ABB RobotStudio station: step_smartcomponet.rspag

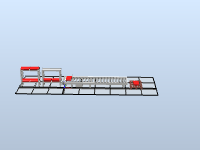
--- station ---
Station step_smartcomponet (saved by RobotStudio 6.8.8307.1040)
Controller IRB_120_3kg_0.58m_3
  mechanical unit ROB_1: IRB120_3_58__01, 6 joints, base frame (0, 0, 0) mm
Layout (positions relative to the parent item):
  - IRB4600_60_205_C_01 [mechanism, from Robots\IRB4600_60_205_C_G_01.rslib] at (0, 0, 0) mm; joint values [0, 0, 0, 0, 0.5236, 0] (rad or m)
  - 950_4000_h2 [part, from Equipment\Conveyor 950 4000 h2.rslib]
  - CAJA [part, from Step_smartcomponet\SOLCAJA.rslib] at (-590.31, 450, 412.42) mm
  - SmartComponent_1 [smart component, from Step_smartcomponet\SmartComponent_1.rslib]
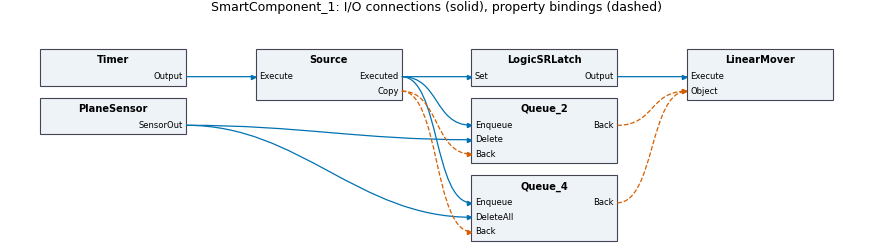
      connections:
        Timer.Output -> Source.Execute
        Source.Executed -> Queue_2.Enqueue
        LogicSRLatch.Output -> LinearMover.Execute
        PlaneSensor.SensorOut -> Queue_2.Delete
        Source.Executed -> Queue_4.Enqueue
        PlaneSensor.SensorOut -> Queue_4.DeleteAll
        Source.Executed -> LogicSRLatch.Set
        Source.Copy => Queue_2.Back
        Queue_2.Back => LinearMover.Object
        Source.Copy => Queue_4.Back
        Queue_4.Back => LinearMover.Object
    - Source [smart component, from Components\Source.rslib]
        properties: Source=CAJA1; Copy=(none); Parent=(none); Position=[3.9 0.5 0.4]; Orientation=[0 0 0]; Transient=true; PhysicsBehavior=0
    - Timer [smart component, from Components\Timer.rslib]
        properties: StartTime=0; Interval=7; Repeat=true; CurrentTime=256.632
    - LinearMover [smart component, from Components\LinearMover.rslib]
        properties: Object=(none); Direction=[-1 0 0]; Speed=0.6; Reference=Global; ReferenceObject=(none)
    - PlaneSensor [smart component, from Components\PlaneSensor.rslib]
        properties: Origin=[0.5 0.1 0.45]; Axis1=[0 0.2 0.3]; Axis2=[0 0.5 0]; SensedPart=(none)
      - _sensorPart_ [part, from Step_smartcomponet\SmartComponent_1.rslib]
    - LogicSRLatch [smart component, from Components\LogicSRLatch.rslib]
    - Queue_4 [smart component, from Components\Queue.rslib]
        properties: Back=(none); Front=(none); Queue={b297857b-f8dc-4992-8a1c-48ad92a09bcc}; NumberOfObjects=1
  - IRB120_3_58__01 [mechanism, from Robots\IRB120_3_58_G_01.rslib] at (0, 0, 0) mm; joint values [0, 0, 0, 0, 0.5236, 0] (rad or m)
  - Plant Shelf Assem [graphiccomponentgroup, from Step_smartcomponet\Stand de cajas vacio.rslib] at (-1309.51, 39.88, -195.16) mm, rotated rx 90 ry 0 rz 90 deg
    - Leg [part, from Step_smartcomponet\Stand de cajas vacio.rslib] at (58.14, 192.19, 978.34) mm, rotated rx 90 ry 0 rz 0 deg
    - Leg [part, from Step_smartcomponet\Stand de cajas vacio.rslib] at (432.79, 192.19, 978.34) mm, rotated rx 90 ry 0 rz 0 deg
    - Leg [part, from Step_smartcomponet\Stand de cajas vacio.rslib] at (58.14, 192.19, -151.96) mm, rotated rx 90 ry 0 rz 0 deg
    - Leg [part, from Step_smartcomponet\Stand de cajas vacio.rslib] at (432.79, 192.19, -151.96) mm, rotated rx 90 ry 0 rz 0 deg
    - Bottom Support Beam [part, from Step_smartcomponet\Stand de cajas vacio.rslib] at (432.79, 395.39, 1016.44) mm, rotated rx 0 ry 90 rz 0 deg
    - Bottom Support Beam [part, from Step_smartcomponet\Stand de cajas vacio.rslib] at (432.79, 395.39, -63.06) mm, rotated rx 0 ry 90 rz 0 deg
    - Top Support Beam [part, from Step_smartcomponet\Stand de cajas vacio.rslib] at (432.79, 1271.69, -63.06) mm, rotated rx 0 ry 90 rz 0 deg
    - Top Support Beam [part, from Step_smartcomponet\Stand de cajas vacio.rslib] at (432.79, 1271.69, 1010.09) mm, rotated rx 0 ry 90 rz 0 deg
    - Shelf Platform [part, from Step_smartcomponet\Stand de cajas vacio.rslib] at (121.64, 1303.08, 1067.24) mm
    - Shelf Platform [part, from Step_smartcomponet\Stand de cajas vacio.rslib] at (216.89, 1303.44, 1067.24) mm
    - Shelf Platform [part, from Step_smartcomponet\Stand de cajas vacio.rslib] at (312.14, 1303.44, 1067.24) mm
    - Shelf Platform [part, from Step_smartcomponet\Stand de cajas vacio.rslib] at (432.79, 1303.44, 1067.24) mm, rotated rx 0 ry 0 rz 90 deg
    - Shelf Platform [part, from Step_smartcomponet\Stand de cajas vacio.rslib] at (96.24, 1398.69, 1067.24) mm, rotated rx 0 ry 0 rz -90 deg
    - Shelf Platform [part, from Step_smartcomponet\Stand de cajas vacio.rslib] at (121.64, 484.29, 1067.24) mm
    - Shelf Platform [part, from Step_smartcomponet\Stand de cajas vacio.rslib] at (216.89, 484.29, 1067.24) mm
    - Shelf Platform [part, from Step_smartcomponet\Stand de cajas vacio.rslib] at (312.14, 484.29, 1067.24) mm
    - Shelf Platform [part, from Step_smartcomponet\Stand de cajas vacio.rslib] at (96.24, 579.54, 1067.24) mm, rotated rx 0 ry 0 rz -90 deg
    - Shelf Platform [part, from Step_smartcomponet\Stand de cajas vacio.rslib] at (432.79, 484.29, 1067.24) mm, rotated rx 0 ry 0 rz 90 deg
    - Bracket [part, from Step_smartcomponet\Stand de cajas vacio.rslib] at (96.24, 395.39, -82.11) mm, rotated rx 90 ry 0 rz 0 deg
    - Bracket [part, from Step_smartcomponet\Stand de cajas vacio.rslib] at (96.24, 1271.69, -78.94) mm, rotated rx 90 ry 0 rz 0 deg
    - Bracket [part, from Step_smartcomponet\Stand de cajas vacio.rslib] at (432.79, 1271.69, -78.94) mm, rotated rx -90 ry 0 rz 180 deg
    - Bracket [part, from Step_smartcomponet\Stand de cajas vacio.rslib] at (432.79, 395.39, -82.11) mm, rotated rx -90 ry 0 rz 180 deg
    - Bracket [part, from Step_smartcomponet\Stand de cajas vacio.rslib] at (96.24, 395.39, 997.39) mm, rotated rx 90 ry 0 rz 0 deg
    - Bracket [part, from Step_smartcomponet\Stand de cajas vacio.rslib] at (96.24, 1271.69, 994.21) mm, rotated rx 90 ry 0 rz 0 deg
    - Bracket [part, from Step_smartcomponet\Stand de cajas vacio.rslib] at (432.79, 1271.69, 994.21) mm, rotated rx -90 ry 0 rz 180 deg
    - Bracket [part, from Step_smartcomponet\Stand de cajas vacio.rslib] at (432.79, 395.39, 997.39) mm, rotated rx -90 ry 0 rz 180 deg
    - 98685A710_BRASS PHILLIPS DECORATIVE ROUNDED HEAD SCREWS [part, from Step_smartcomponet\Stand de cajas vacio.rslib] at (109.47, 1276.01, -78.94) mm, rotated rx 0 ry 0 rz 90 deg
    - 98685A710_BRASS PHILLIPS DECORATIVE ROUNDED HEAD SCREWS [part, from Step_smartcomponet\Stand de cajas vacio.rslib] at (419.57, 1276.01, -78.94) mm, rotated rx 180 ry 0 rz 90 deg
    - 98685A710_BRASS PHILLIPS DECORATIVE ROUNDED HEAD SCREWS [part, from Step_smartcomponet\Stand de cajas vacio.rslib] at (91.93, 1260.06, -78.94) mm, rotated rx 67.55 ry 0 rz 180 deg
    - 98685A710_BRASS PHILLIPS DECORATIVE ROUNDED HEAD SCREWS [part, from Step_smartcomponet\Stand de cajas vacio.rslib] at (437.11, 1260.06, -78.94) mm, rotated rx 112.45 ry 0 rz 0 deg
    - 98685A710_BRASS PHILLIPS DECORATIVE ROUNDED HEAD SCREWS [part, from Step_smartcomponet\Stand de cajas vacio.rslib] at (109.47, 1276.01, 994.21) mm, rotated rx -16.06 ry 0 rz 90 deg
    - 98685A710_BRASS PHILLIPS DECORATIVE ROUNDED HEAD SCREWS [part, from Step_smartcomponet\Stand de cajas vacio.rslib] at (419.57, 1276.01, 994.21) mm, rotated rx -163.94 ry 0 rz 90 deg
    - 98685A710_BRASS PHILLIPS DECORATIVE ROUNDED HEAD SCREWS [part, from Step_smartcomponet\Stand de cajas vacio.rslib] at (91.93, 1260.06, 994.21) mm, rotated rx -112.45 ry 0 rz 180 deg
    - 98685A710_BRASS PHILLIPS DECORATIVE ROUNDED HEAD SCREWS [part, from Step_smartcomponet\Stand de cajas vacio.rslib] at (437.11, 1260.07, 994.21) mm, rotated rx -67.55 ry 0 rz 0 deg
    - 98685A710_BRASS PHILLIPS DECORATIVE ROUNDED HEAD SCREWS [part, from Step_smartcomponet\Stand de cajas vacio.rslib] at (91.93, 383.76, 997.39) mm, rotated rx -112.45 ry 0 rz 180 deg
    - 98685A710_BRASS PHILLIPS DECORATIVE ROUNDED HEAD SCREWS [part, from Step_smartcomponet\Stand de cajas vacio.rslib] at (437.11, 383.77, 997.39) mm, rotated rx -67.55 ry 0 rz 0 deg
    - 98685A710_BRASS PHILLIPS DECORATIVE ROUNDED HEAD SCREWS [part, from Step_smartcomponet\Stand de cajas vacio.rslib] at (109.47, 399.71, 997.39) mm, rotated rx 0 ry 0 rz 90 deg
    - 98685A710_BRASS PHILLIPS DECORATIVE ROUNDED HEAD SCREWS [part, from Step_smartcomponet\Stand de cajas vacio.rslib] at (419.57, 399.71, 997.38) mm, rotated rx 180 ry 0 rz 90 deg
    - 98685A710_BRASS PHILLIPS DECORATIVE ROUNDED HEAD SCREWS [part, from Step_smartcomponet\Stand de cajas vacio.rslib] at (109.47, 399.71, -82.11) mm, rotated rx 0 ry 0 rz 90 deg
    - 98685A710_BRASS PHILLIPS DECORATIVE ROUNDED HEAD SCREWS [part, from Step_smartcomponet\Stand de cajas vacio.rslib] at (419.57, 399.71, -82.12) mm, rotated rx 180 ry 0 rz 90 deg
    - 98685A710_BRASS PHILLIPS DECORATIVE ROUNDED HEAD SCREWS [part, from Step_smartcomponet\Stand de cajas vacio.rslib] at (91.93, 383.76, -82.11) mm, rotated rx -112.45 ry 0 rz 180 deg
    - 98685A710_BRASS PHILLIPS DECORATIVE ROUNDED HEAD SCREWS [part, from Step_smartcomponet\Stand de cajas vacio.rslib] at (437.11, 383.77, -82.11) mm, rotated rx -67.55 ry 0 rz 0 deg
    - 90294A157_PHILLIPS FLAT HEAD SCREWS FOR WOOD [part, from Step_smartcomponet\Stand de cajas vacio.rslib] at (426.87, 1366.94, 994.21) mm
    - 90294A157_PHILLIPS FLAT HEAD SCREWS FOR WOOD [part, from Step_smartcomponet\Stand de cajas vacio.rslib] at (426.87, 1335.19, 994.21) mm
    - 90294A157_PHILLIPS FLAT HEAD SCREWS FOR WOOD [part, from Step_smartcomponet\Stand de cajas vacio.rslib] at (375.64, 1309.36, 994.21) mm, rotated rx 0 ry 0 rz -90 deg
    - 90294A157_PHILLIPS FLAT HEAD SCREWS FOR WOOD [part, from Step_smartcomponet\Stand de cajas vacio.rslib] at (343.89, 1309.36, 994.21) mm, rotated rx 0 ry 0 rz -90 deg
    - 90294A157_PHILLIPS FLAT HEAD SCREWS FOR WOOD [part, from Step_smartcomponet\Stand de cajas vacio.rslib] at (280.39, 1309.36, 994.21) mm, rotated rx 0 ry 0 rz -90 deg
    - 90294A157_PHILLIPS FLAT HEAD SCREWS FOR WOOD [part, from Step_smartcomponet\Stand de cajas vacio.rslib] at (248.64, 1309.36, 994.21) mm, rotated rx 0 ry 0 rz -90 deg
    - 90294A157_PHILLIPS FLAT HEAD SCREWS FOR WOOD [part, from Step_smartcomponet\Stand de cajas vacio.rslib] at (185.14, 1309, 994.21) mm, rotated rx 0 ry 0 rz -90 deg
    - 90294A157_PHILLIPS FLAT HEAD SCREWS FOR WOOD [part, from Step_smartcomponet\Stand de cajas vacio.rslib] at (153.39, 1309, 994.21) mm, rotated rx 0 ry 0 rz -90 deg
    - 90294A157_PHILLIPS FLAT HEAD SCREWS FOR WOOD [part, from Step_smartcomponet\Stand de cajas vacio.rslib] at (102.16, 1335.19, 994.21) mm, rotated rx 67.55 ry 0 rz 180 deg
    - 90294A157_PHILLIPS FLAT HEAD SCREWS FOR WOOD [part, from Step_smartcomponet\Stand de cajas vacio.rslib] at (102.16, 1366.94, 994.21) mm, rotated rx 67.55 ry 0 rz 180 deg
    - 90294A157_PHILLIPS FLAT HEAD SCREWS FOR WOOD [part, from Step_smartcomponet\Stand de cajas vacio.rslib] at (102.16, 516.04, 994.21) mm, rotated rx 67.55 ry 0 rz 180 deg
    - 90294A157_PHILLIPS FLAT HEAD SCREWS FOR WOOD [part, from Step_smartcomponet\Stand de cajas vacio.rslib] at (153.39, 490.21, 994.21) mm, rotated rx 0 ry 0 rz -90 deg
    - 90294A157_PHILLIPS FLAT HEAD SCREWS FOR WOOD [part, from Step_smartcomponet\Stand de cajas vacio.rslib] at (426.87, 516.04, 994.21) mm
    - 90294A157_PHILLIPS FLAT HEAD SCREWS FOR WOOD [part, from Step_smartcomponet\Stand de cajas vacio.rslib] at (426.87, 547.79, 994.21) mm
    - 90294A157_PHILLIPS FLAT HEAD SCREWS FOR WOOD [part, from Step_smartcomponet\Stand de cajas vacio.rslib] at (343.89, 490.21, 994.21) mm, rotated rx 0 ry 0 rz -90 deg
    - 90294A157_PHILLIPS FLAT HEAD SCREWS FOR WOOD [part, from Step_smartcomponet\Stand de cajas vacio.rslib] at (375.64, 490.21, 994.21) mm, rotated rx 0 ry 0 rz -90 deg
    - 90294A157_PHILLIPS FLAT HEAD SCREWS FOR WOOD [part, from Step_smartcomponet\Stand de cajas vacio.rslib] at (248.64, 490.21, 994.21) mm, rotated rx 0 ry 0 rz -90 deg
    - 90294A157_PHILLIPS FLAT HEAD SCREWS FOR WOOD [part, from Step_smartcomponet\Stand de cajas vacio.rslib] at (280.39, 490.21, 994.21) mm, rotated rx 0 ry 0 rz -90 deg
    - 90294A157_PHILLIPS FLAT HEAD SCREWS FOR WOOD [part, from Step_smartcomponet\Stand de cajas vacio.rslib] at (102.16, 547.79, 994.21) mm, rotated rx 67.55 ry 0 rz 180 deg
    - 90294A157_PHILLIPS FLAT HEAD SCREWS FOR WOOD [part, from Step_smartcomponet\Stand de cajas vacio.rslib] at (185.14, 490.21, 994.21) mm, rotated rx 0 ry 0 rz -90 deg
    - 90294A157_PHILLIPS FLAT HEAD SCREWS FOR WOOD [part, from Step_smartcomponet\Stand de cajas vacio.rslib] at (426.87, 1366.94, -78.94) mm
    - 90294A157_PHILLIPS FLAT HEAD SCREWS FOR WOOD [part, from Step_smartcomponet\Stand de cajas vacio.rslib] at (426.87, 1335.19, -78.94) mm
    - 90294A157_PHILLIPS FLAT HEAD SCREWS FOR WOOD [part, from Step_smartcomponet\Stand de cajas vacio.rslib] at (375.64, 1309.36, -78.94) mm, rotated rx 0 ry 0 rz -90 deg
    - 90294A157_PHILLIPS FLAT HEAD SCREWS FOR WOOD [part, from Step_smartcomponet\Stand de cajas vacio.rslib] at (343.89, 1309.36, -78.94) mm, rotated rx 0 ry 0 rz -90 deg
    - 90294A157_PHILLIPS FLAT HEAD SCREWS FOR WOOD [part, from Step_smartcomponet\Stand de cajas vacio.rslib] at (280.39, 1309.36, -78.94) mm, rotated rx 0 ry 0 rz -90 deg
    - 90294A157_PHILLIPS FLAT HEAD SCREWS FOR WOOD [part, from Step_smartcomponet\Stand de cajas vacio.rslib] at (248.64, 1309.36, -78.94) mm, rotated rx 0 ry 0 rz -90 deg
    - 90294A157_PHILLIPS FLAT HEAD SCREWS FOR WOOD [part, from Step_smartcomponet\Stand de cajas vacio.rslib] at (185.14, 1309, -78.94) mm, rotated rx 0 ry 0 rz -90 deg
    - 90294A157_PHILLIPS FLAT HEAD SCREWS FOR WOOD [part, from Step_smartcomponet\Stand de cajas vacio.rslib] at (153.39, 1309, -78.94) mm, rotated rx 0 ry 0 rz -90 deg
    - 90294A157_PHILLIPS FLAT HEAD SCREWS FOR WOOD [part, from Step_smartcomponet\Stand de cajas vacio.rslib] at (102.16, 1335.19, -78.94) mm, rotated rx -67.55 ry 0 rz 180 deg
    - 90294A157_PHILLIPS FLAT HEAD SCREWS FOR WOOD [part, from Step_smartcomponet\Stand de cajas vacio.rslib] at (102.16, 1366.94, -78.94) mm, rotated rx -67.55 ry 0 rz 180 deg
    - 90294A157_PHILLIPS FLAT HEAD SCREWS FOR WOOD [part, from Step_smartcomponet\Stand de cajas vacio.rslib] at (102.16, 516.04, -78.94) mm, rotated rx -67.55 ry 0 rz 180 deg
    - 90294A157_PHILLIPS FLAT HEAD SCREWS FOR WOOD [part, from Step_smartcomponet\Stand de cajas vacio.rslib] at (153.39, 490.21, -78.94) mm, rotated rx 0 ry 0 rz -90 deg
    - 90294A157_PHILLIPS FLAT HEAD SCREWS FOR WOOD [part, from Step_smartcomponet\Stand de cajas vacio.rslib] at (426.87, 516.04, -78.94) mm
    - 90294A157_PHILLIPS FLAT HEAD SCREWS FOR WOOD [part, from Step_smartcomponet\Stand de cajas vacio.rslib] at (426.87, 547.79, -78.94) mm
    - 90294A157_PHILLIPS FLAT HEAD SCREWS FOR WOOD [part, from Step_smartcomponet\Stand de cajas vacio.rslib] at (343.89, 490.21, -78.94) mm, rotated rx 0 ry 0 rz -90 deg
    - 90294A157_PHILLIPS FLAT HEAD SCREWS FOR WOOD [part, from Step_smartcomponet\Stand de cajas vacio.rslib] at (375.64, 490.21, -78.94) mm, rotated rx 0 ry 0 rz -90 deg
    - 90294A157_PHILLIPS FLAT HEAD SCREWS FOR WOOD [part, from Step_smartcomponet\Stand de cajas vacio.rslib] at (248.64, 490.21, -78.94) mm, rotated rx 0 ry 0 rz -90 deg
    - 90294A157_PHILLIPS FLAT HEAD SCREWS FOR WOOD [part, from Step_smartcomponet\Stand de cajas vacio.rslib] at (280.39, 490.21, -78.94) mm, rotated rx 0 ry 0 rz -90 deg
    - 90294A157_PHILLIPS FLAT HEAD SCREWS FOR WOOD [part, from Step_smartcomponet\Stand de cajas vacio.rslib] at (102.16, 547.79, -78.94) mm, rotated rx -67.55 ry 0 rz 180 deg
    - 90294A157_PHILLIPS FLAT HEAD SCREWS FOR WOOD [part, from Step_smartcomponet\Stand de cajas vacio.rslib] at (185.14, 490.21, -78.94) mm, rotated rx 0 ry 0 rz -90 deg
  - Plant Shelf Assem_2 [graphiccomponentgroup, from Step_smartcomponet\Stand de cajas vacio.rslib] at (-2715.59, 39.88, -195.16) mm, rotated rx 90 ry 0 rz 90 deg
    - Leg [part, from Step_smartcomponet\Stand de cajas vacio.rslib] at (58.14, 192.19, 978.34) mm, rotated rx 90 ry 0 rz 0 deg
    - Leg [part, from Step_smartcomponet\Stand de cajas vacio.rslib] at (432.79, 192.19, 978.34) mm, rotated rx 90 ry 0 rz 0 deg
    - Leg [part, from Step_smartcomponet\Stand de cajas vacio.rslib] at (58.14, 192.19, -151.96) mm, rotated rx 90 ry 0 rz 0 deg
    - Leg [part, from Step_smartcomponet\Stand de cajas vacio.rslib] at (432.79, 192.19, -151.96) mm, rotated rx 90 ry 0 rz 0 deg
    - Bottom Support Beam [part, from Step_smartcomponet\Stand de cajas vacio.rslib] at (432.79, 395.39, 1016.44) mm, rotated rx 0 ry 90 rz 0 deg
    - Bottom Support Beam [part, from Step_smartcomponet\Stand de cajas vacio.rslib] at (432.79, 395.39, -63.06) mm, rotated rx 0 ry 90 rz 0 deg
    - Top Support Beam [part, from Step_smartcomponet\Stand de cajas vacio.rslib] at (432.79, 1271.69, -63.06) mm, rotated rx 0 ry 90 rz 0 deg
    - Top Support Beam [part, from Step_smartcomponet\Stand de cajas vacio.rslib] at (432.79, 1271.69, 1010.09) mm, rotated rx 0 ry 90 rz 0 deg
    - Shelf Platform [part, from Step_smartcomponet\Stand de cajas vacio.rslib] at (121.64, 1303.08, 1067.24) mm
    - Shelf Platform [part, from Step_smartcomponet\Stand de cajas vacio.rslib] at (216.89, 1303.44, 1067.24) mm
    - Shelf Platform [part, from Step_smartcomponet\Stand de cajas vacio.rslib] at (312.14, 1303.44, 1067.24) mm
    - Shelf Platform [part, from Step_smartcomponet\Stand de cajas vacio.rslib] at (432.79, 1303.44, 1067.24) mm, rotated rx 0 ry 0 rz 90 deg
    - Shelf Platform [part, from Step_smartcomponet\Stand de cajas vacio.rslib] at (96.24, 1398.69, 1067.24) mm, rotated rx 0 ry 0 rz -90 deg
    - Shelf Platform [part, from Step_smartcomponet\Stand de cajas vacio.rslib] at (121.64, 484.29, 1067.24) mm
    - Shelf Platform [part, from Step_smartcomponet\Stand de cajas vacio.rslib] at (216.89, 484.29, 1067.24) mm
    - Shelf Platform [part, from Step_smartcomponet\Stand de cajas vacio.rslib] at (312.14, 484.29, 1067.24) mm
    - Shelf Platform [part, from Step_smartcomponet\Stand de cajas vacio.rslib] at (96.24, 579.54, 1067.24) mm, rotated rx 0 ry 0 rz -90 deg
    - Shelf Platform [part, from Step_smartcomponet\Stand de cajas vacio.rslib] at (432.79, 484.29, 1067.24) mm, rotated rx 0 ry 0 rz 90 deg
    - Bracket [part, from Step_smartcomponet\Stand de cajas vacio.rslib] at (96.24, 395.39, -82.11) mm, rotated rx 90 ry 0 rz 0 deg
    - Bracket [part, from Step_smartcomponet\Stand de cajas vacio.rslib] at (96.24, 1271.69, -78.94) mm, rotated rx 90 ry 0 rz 0 deg
    - Bracket [part, from Step_smartcomponet\Stand de cajas vacio.rslib] at (432.79, 1271.69, -78.94) mm, rotated rx -90 ry 0 rz 180 deg
    - Bracket [part, from Step_smartcomponet\Stand de cajas vacio.rslib] at (432.79, 395.39, -82.11) mm, rotated rx -90 ry 0 rz 180 deg
    - Bracket [part, from Step_smartcomponet\Stand de cajas vacio.rslib] at (96.24, 395.39, 997.39) mm, rotated rx 90 ry 0 rz 0 deg
    - Bracket [part, from Step_smartcomponet\Stand de cajas vacio.rslib] at (96.24, 1271.69, 994.21) mm, rotated rx 90 ry 0 rz 0 deg
    - Bracket [part, from Step_smartcomponet\Stand de cajas vacio.rslib] at (432.79, 1271.69, 994.21) mm, rotated rx -90 ry 0 rz 180 deg
    - Bracket [part, from Step_smartcomponet\Stand de cajas vacio.rslib] at (432.79, 395.39, 997.39) mm, rotated rx -90 ry 0 rz 180 deg
    - 98685A710_BRASS PHILLIPS DECORATIVE ROUNDED HEAD SCREWS [part, from Step_smartcomponet\Stand de cajas vacio.rslib] at (109.47, 1276.01, -78.94) mm, rotated rx 0 ry 0 rz 90 deg
    - 98685A710_BRASS PHILLIPS DECORATIVE ROUNDED HEAD SCREWS [part, from Step_smartcomponet\Stand de cajas vacio.rslib] at (419.57, 1276.01, -78.94) mm, rotated rx 180 ry 0 rz 90 deg
    - 98685A710_BRASS PHILLIPS DECORATIVE ROUNDED HEAD SCREWS [part, from Step_smartcomponet\Stand de cajas vacio.rslib] at (91.93, 1260.06, -78.94) mm, rotated rx 67.55 ry 0 rz 180 deg
    - 98685A710_BRASS PHILLIPS DECORATIVE ROUNDED HEAD SCREWS [part, from Step_smartcomponet\Stand de cajas vacio.rslib] at (437.11, 1260.06, -78.94) mm, rotated rx 112.45 ry 0 rz 0 deg
    - 98685A710_BRASS PHILLIPS DECORATIVE ROUNDED HEAD SCREWS [part, from Step_smartcomponet\Stand de cajas vacio.rslib] at (109.47, 1276.01, 994.21) mm, rotated rx -16.06 ry 0 rz 90 deg
    - 98685A710_BRASS PHILLIPS DECORATIVE ROUNDED HEAD SCREWS [part, from Step_smartcomponet\Stand de cajas vacio.rslib] at (419.57, 1276.01, 994.21) mm, rotated rx -163.94 ry 0 rz 90 deg
    - 98685A710_BRASS PHILLIPS DECORATIVE ROUNDED HEAD SCREWS [part, from Step_smartcomponet\Stand de cajas vacio.rslib] at (91.93, 1260.06, 994.21) mm, rotated rx -112.45 ry 0 rz 180 deg
    - 98685A710_BRASS PHILLIPS DECORATIVE ROUNDED HEAD SCREWS [part, from Step_smartcomponet\Stand de cajas vacio.rslib] at (437.11, 1260.07, 994.21) mm, rotated rx -67.55 ry 0 rz 0 deg
    - 98685A710_BRASS PHILLIPS DECORATIVE ROUNDED HEAD SCREWS [part, from Step_smartcomponet\Stand de cajas vacio.rslib] at (91.93, 383.76, 997.39) mm, rotated rx -112.45 ry 0 rz 180 deg
    - 98685A710_BRASS PHILLIPS DECORATIVE ROUNDED HEAD SCREWS [part, from Step_smartcomponet\Stand de cajas vacio.rslib] at (437.11, 383.77, 997.39) mm, rotated rx -67.55 ry 0 rz 0 deg
    - 98685A710_BRASS PHILLIPS DECORATIVE ROUNDED HEAD SCREWS [part, from Step_smartcomponet\Stand de cajas vacio.rslib] at (109.47, 399.71, 997.39) mm, rotated rx 0 ry 0 rz 90 deg
    - 98685A710_BRASS PHILLIPS DECORATIVE ROUNDED HEAD SCREWS [part, from Step_smartcomponet\Stand de cajas vacio.rslib] at (419.57, 399.71, 997.38) mm, rotated rx 180 ry 0 rz 90 deg
    - 98685A710_BRASS PHILLIPS DECORATIVE ROUNDED HEAD SCREWS [part, from Step_smartcomponet\Stand de cajas vacio.rslib] at (109.47, 399.71, -82.11) mm, rotated rx 0 ry 0 rz 90 deg
    - 98685A710_BRASS PHILLIPS DECORATIVE ROUNDED HEAD SCREWS [part, from Step_smartcomponet\Stand de cajas vacio.rslib] at (419.57, 399.71, -82.12) mm, rotated rx 180 ry 0 rz 90 deg
    - 98685A710_BRASS PHILLIPS DECORATIVE ROUNDED HEAD SCREWS [part, from Step_smartcomponet\Stand de cajas vacio.rslib] at (91.93, 383.76, -82.11) mm, rotated rx -112.45 ry 0 rz 180 deg
    - 98685A710_BRASS PHILLIPS DECORATIVE ROUNDED HEAD SCREWS [part, from Step_smartcomponet\Stand de cajas vacio.rslib] at (437.11, 383.77, -82.11) mm, rotated rx -67.55 ry 0 rz 0 deg
    - 90294A157_PHILLIPS FLAT HEAD SCREWS FOR WOOD [part, from Step_smartcomponet\Stand de cajas vacio.rslib] at (426.87, 1366.94, 994.21) mm
    - 90294A157_PHILLIPS FLAT HEAD SCREWS FOR WOOD [part, from Step_smartcomponet\Stand de cajas vacio.rslib] at (426.87, 1335.19, 994.21) mm
    - 90294A157_PHILLIPS FLAT HEAD SCREWS FOR WOOD [part, from Step_smartcomponet\Stand de cajas vacio.rslib] at (375.64, 1309.36, 994.21) mm, rotated rx 0 ry 0 rz -90 deg
    - 90294A157_PHILLIPS FLAT HEAD SCREWS FOR WOOD [part, from Step_smartcomponet\Stand de cajas vacio.rslib] at (343.89, 1309.36, 994.21) mm, rotated rx 0 ry 0 rz -90 deg
    - 90294A157_PHILLIPS FLAT HEAD SCREWS FOR WOOD [part, from Step_smartcomponet\Stand de cajas vacio.rslib] at (280.39, 1309.36, 994.21) mm, rotated rx 0 ry 0 rz -90 deg
    - 90294A157_PHILLIPS FLAT HEAD SCREWS FOR WOOD [part, from Step_smartcomponet\Stand de cajas vacio.rslib] at (248.64, 1309.36, 994.21) mm, rotated rx 0 ry 0 rz -90 deg
    - 90294A157_PHILLIPS FLAT HEAD SCREWS FOR WOOD [part, from Step_smartcomponet\Stand de cajas vacio.rslib] at (185.14, 1309, 994.21) mm, rotated rx 0 ry 0 rz -90 deg
    - 90294A157_PHILLIPS FLAT HEAD SCREWS FOR WOOD [part, from Step_smartcomponet\Stand de cajas vacio.rslib] at (153.39, 1309, 994.21) mm, rotated rx 0 ry 0 rz -90 deg
    - 90294A157_PHILLIPS FLAT HEAD SCREWS FOR WOOD [part, from Step_smartcomponet\Stand de cajas vacio.rslib] at (102.16, 1335.19, 994.21) mm, rotated rx 67.55 ry 0 rz 180 deg
    - 90294A157_PHILLIPS FLAT HEAD SCREWS FOR WOOD [part, from Step_smartcomponet\Stand de cajas vacio.rslib] at (102.16, 1366.94, 994.21) mm, rotated rx 67.55 ry 0 rz 180 deg
    - 90294A157_PHILLIPS FLAT HEAD SCREWS FOR WOOD [part, from Step_smartcomponet\Stand de cajas vacio.rslib] at (102.16, 516.04, 994.21) mm, rotated rx 67.55 ry 0 rz 180 deg
    - 90294A157_PHILLIPS FLAT HEAD SCREWS FOR WOOD [part, from Step_smartcomponet\Stand de cajas vacio.rslib] at (153.39, 490.21, 994.21) mm, rotated rx 0 ry 0 rz -90 deg
    - 90294A157_PHILLIPS FLAT HEAD SCREWS FOR WOOD [part, from Step_smartcomponet\Stand de cajas vacio.rslib] at (426.87, 516.04, 994.21) mm
    - 90294A157_PHILLIPS FLAT HEAD SCREWS FOR WOOD [part, from Step_smartcomponet\Stand de cajas vacio.rslib] at (426.87, 547.79, 994.21) mm
    - 90294A157_PHILLIPS FLAT HEAD SCREWS FOR WOOD [part, from Step_smartcomponet\Stand de cajas vacio.rslib] at (343.89, 490.21, 994.21) mm, rotated rx 0 ry 0 rz -90 deg
    - 90294A157_PHILLIPS FLAT HEAD SCREWS FOR WOOD [part, from Step_smartcomponet\Stand de cajas vacio.rslib] at (375.64, 490.21, 994.21) mm, rotated rx 0 ry 0 rz -90 deg
    - 90294A157_PHILLIPS FLAT HEAD SCREWS FOR WOOD [part, from Step_smartcomponet\Stand de cajas vacio.rslib] at (248.64, 490.21, 994.21) mm, rotated rx 0 ry 0 rz -90 deg
    - 90294A157_PHILLIPS FLAT HEAD SCREWS FOR WOOD [part, from Step_smartcomponet\Stand de cajas vacio.rslib] at (280.39, 490.21, 994.21) mm, rotated rx 0 ry 0 rz -90 deg
    - 90294A157_PHILLIPS FLAT HEAD SCREWS FOR WOOD [part, from Step_smartcomponet\Stand de cajas vacio.rslib] at (102.16, 547.79, 994.21) mm, rotated rx 67.55 ry 0 rz 180 deg
    - 90294A157_PHILLIPS FLAT HEAD SCREWS FOR WOOD [part, from Step_smartcomponet\Stand de cajas vacio.rslib] at (185.14, 490.21, 994.21) mm, rotated rx 0 ry 0 rz -90 deg
    - 90294A157_PHILLIPS FLAT HEAD SCREWS FOR WOOD [part, from Step_smartcomponet\Stand de cajas vacio.rslib] at (426.87, 1366.94, -78.94) mm
    - 90294A157_PHILLIPS FLAT HEAD SCREWS FOR WOOD [part, from Step_smartcomponet\Stand de cajas vacio.rslib] at (426.87, 1335.19, -78.94) mm
    - 90294A157_PHILLIPS FLAT HEAD SCREWS FOR WOOD [part, from Step_smartcomponet\Stand de cajas vacio.rslib] at (375.64, 1309.36, -78.94) mm, rotated rx 0 ry 0 rz -90 deg
    - 90294A157_PHILLIPS FLAT HEAD SCREWS FOR WOOD [part, from Step_smartcomponet\Stand de cajas vacio.rslib] at (343.89, 1309.36, -78.94) mm, rotated rx 0 ry 0 rz -90 deg
    - 90294A157_PHILLIPS FLAT HEAD SCREWS FOR WOOD [part, from Step_smartcomponet\Stand de cajas vacio.rslib] at (280.39, 1309.36, -78.94) mm, rotated rx 0 ry 0 rz -90 deg
    - 90294A157_PHILLIPS FLAT HEAD SCREWS FOR WOOD [part, from Step_smartcomponet\Stand de cajas vacio.rslib] at (248.64, 1309.36, -78.94) mm, rotated rx 0 ry 0 rz -90 deg
    - 90294A157_PHILLIPS FLAT HEAD SCREWS FOR WOOD [part, from Step_smartcomponet\Stand de cajas vacio.rslib] at (185.14, 1309, -78.94) mm, rotated rx 0 ry 0 rz -90 deg
    - 90294A157_PHILLIPS FLAT HEAD SCREWS FOR WOOD [part, from Step_smartcomponet\Stand de cajas vacio.rslib] at (153.39, 1309, -78.94) mm, rotated rx 0 ry 0 rz -90 deg
    - 90294A157_PHILLIPS FLAT HEAD SCREWS FOR WOOD [part, from Step_smartcomponet\Stand de cajas vacio.rslib] at (102.16, 1335.19, -78.94) mm, rotated rx -67.55 ry 0 rz 180 deg
    - 90294A157_PHILLIPS FLAT HEAD SCREWS FOR WOOD [part, from Step_smartcomponet\Stand de cajas vacio.rslib] at (102.16, 1366.94, -78.94) mm, rotated rx -67.55 ry 0 rz 180 deg
    - 90294A157_PHILLIPS FLAT HEAD SCREWS FOR WOOD [part, from Step_smartcomponet\Stand de cajas vacio.rslib] at (102.16, 516.04, -78.94) mm, rotated rx -67.55 ry 0 rz 180 deg
    - 90294A157_PHILLIPS FLAT HEAD SCREWS FOR WOOD [part, from Step_smartcomponet\Stand de cajas vacio.rslib] at (153.39, 490.21, -78.94) mm, rotated rx 0 ry 0 rz -90 deg
    - 90294A157_PHILLIPS FLAT HEAD SCREWS FOR WOOD [part, from Step_smartcomponet\Stand de cajas vacio.rslib] at (426.87, 516.04, -78.94) mm
    - 90294A157_PHILLIPS FLAT HEAD SCREWS FOR WOOD [part, from Step_smartcomponet\Stand de cajas vacio.rslib] at (426.87, 547.79, -78.94) mm
    - 90294A157_PHILLIPS FLAT HEAD SCREWS FOR WOOD [part, from Step_smartcomponet\Stand de cajas vacio.rslib] at (343.89, 490.21, -78.94) mm, rotated rx 0 ry 0 rz -90 deg
    - 90294A157_PHILLIPS FLAT HEAD SCREWS FOR WOOD [part, from Step_smartcomponet\Stand de cajas vacio.rslib] at (375.64, 490.21, -78.94) mm, rotated rx 0 ry 0 rz -90 deg
    - 90294A157_PHILLIPS FLAT HEAD SCREWS FOR WOOD [part, from Step_smartcomponet\Stand de cajas vacio.rslib] at (248.64, 490.21, -78.94) mm, rotated rx 0 ry 0 rz -90 deg
    - 90294A157_PHILLIPS FLAT HEAD SCREWS FOR WOOD [part, from Step_smartcomponet\Stand de cajas vacio.rslib] at (280.39, 490.21, -78.94) mm, rotated rx 0 ry 0 rz -90 deg
    - 90294A157_PHILLIPS FLAT HEAD SCREWS FOR WOOD [part, from Step_smartcomponet\Stand de cajas vacio.rslib] at (102.16, 547.79, -78.94) mm, rotated rx -67.55 ry 0 rz 180 deg
    - 90294A157_PHILLIPS FLAT HEAD SCREWS FOR WOOD [part, from Step_smartcomponet\Stand de cajas vacio.rslib] at (185.14, 490.21, -78.94) mm, rotated rx 0 ry 0 rz -90 deg
  - Euro Pallet [graphiccomponentgroup, from Equipment\Euro Pallet.rslib] at (5096.44, -117.51, -9.34) mm, rotated rx 0 ry 0 rz 90 deg
    - Body 1 [part, from Equipment\Euro Pallet.rslib]
  - CAJA1 [part, from Step_smartcomponet\SOLCAJA.rslib] at (3859.03, 457.12, 108.49) mm
  - CAJA_2 [part, from Step_smartcomponet\SOLCAJA.rslib] at (-1164.03, -557.08, 357.98) mm, rotated rx 0 ry 0 rz 90 deg
  - CAJA_3 [part, from Step_smartcomponet\SOLCAJA.rslib] at (-546.46, -548.72, 358.29) mm, rotated rx 0 ry 0 rz 90 deg
  - CAJA_4 [part, from Step_smartcomponet\SOLCAJA.rslib] at (-2554.39, -550.04, 315.08) mm, rotated rx 0 ry 0 rz 90 deg
  - CAJA_5 [part, from Step_smartcomponet\SOLCAJA.rslib] at (-1974.28, -548.3, 318.37) mm, rotated rx 0 ry 0 rz 90 deg
  - CAJA_6 [part, from Step_smartcomponet\SOLCAJA.rslib] at (-1950.77, -538.39, 1145.55) mm, rotated rx 0 ry 0 rz 90 deg
  - CAJA_7 [part, from Step_smartcomponet\SOLCAJA.rslib] at (-2559.7, -535.8, 1144) mm, rotated rx 0 ry 0 rz 90 deg

--- Backups/IRB_120_3kg_0.58m_3/RAPID/TASK1/PROGMOD/Module1.mod ---
MODULE Module1
    !***********************************************************
    !
    ! Module:  Module1
    !
    ! Description:
    !   <Insert description here>
    !
    ! Author: Elida Dominguez
    !
    ! Version: 1.0
    !
    !***********************************************************


    !***********************************************************
    !
    ! Procedure main
    !
    !   This is the entry point of your program
    !
    !***********************************************************
    PROC main()
        !Add your code here
    ENDPROC
ENDMODULE
